// TIA Portal V18 export
FUNCTION "fpd_magnet_lightbarrier_main" : Void   // FC3, FBD
{ S7_Optimized_Access := 'TRUE' }
VERSION : 0.1
// stored: AutoNumber true, IsIECCheckEnabled false, SetENOAutomatically false, UDAEnableTagReadback false
   VAR_TEMP
      er_no_clos : Bool;
      er_no_opn : Bool;
      er_both_sensors : Bool;
   END_VAR
BEGIN

REGION Network 1
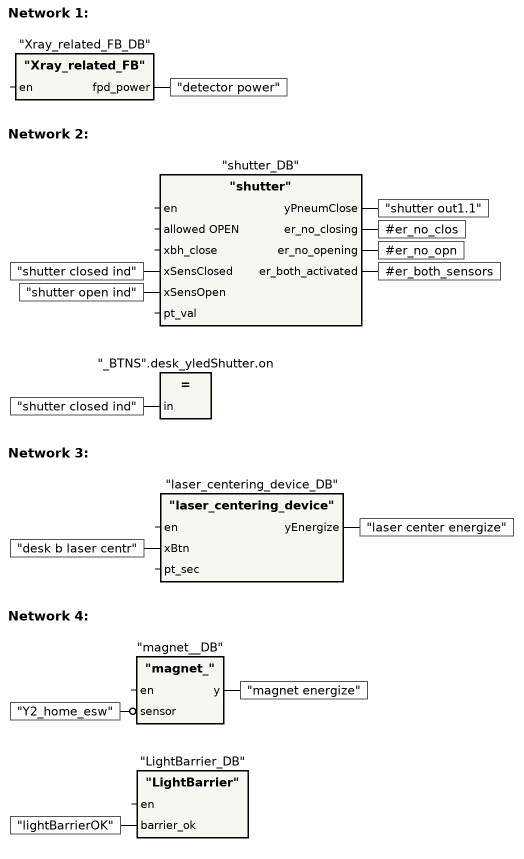
   "Xray_related_FB_DB"(fpd_power => "detector power");   // "Xray_related_FB"
END_REGION

REGION Network 2
   "shutter_DB"(xSensClosed := "shutter closed ind",   // "shutter"
                xSensOpen := "shutter open ind",
                yPneumClose => "shutter out1.1",
                er_no_closing => #er_no_clos,
                er_no_opening => #er_no_opn,
                er_both_activated => #er_both_sensors);
   "_BTNS".desk_yledShutter.on := "shutter closed ind";
END_REGION

REGION Network 3
   "laser_centering_device_DB"(xBtn := "desk b laser centr", yEnergize => "laser center energize");   // "laser_centering_device"
END_REGION

REGION Network 4
   "magnet__DB"(sensor := NOT "Y2_home_esw", y => "magnet energize");   // "magnet_"
   "LightBarrier_DB"(barrier_ok := "lightBarrierOK");   // "LightBarrier"
END_REGION

REGION Network 5
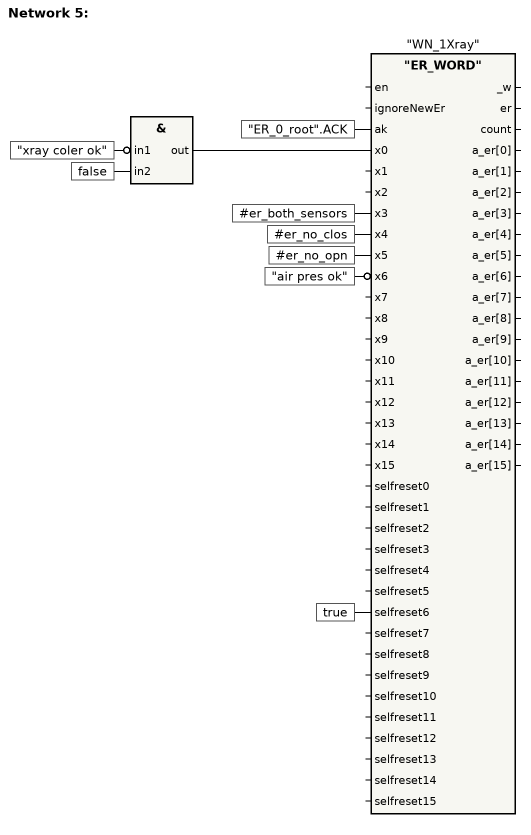
   "WN_1Xray"(ak := "ER_0_root".ACK,   // "ER_WORD"
              x0 := NOT "xray coler ok" AND false,
              x3 := #er_both_sensors,
              x4 := #er_no_clos,
              x5 := #er_no_opn,
              x6 := NOT "air pres ok",
              selfreset6 := true);
END_REGION
END_FUNCTION
